PROGRAM main
VAR
    CountPulse AT %QX0.0 : BOOL;
    ResetCounter AT %QX0.1 : BOOL;
    Done AT %QX0.2 : BOOL;
    CurrentCount AT %MD0 : DINT;

    CounterInstance : CTU_DINT;
    Preset : DINT := 3;
END_VAR

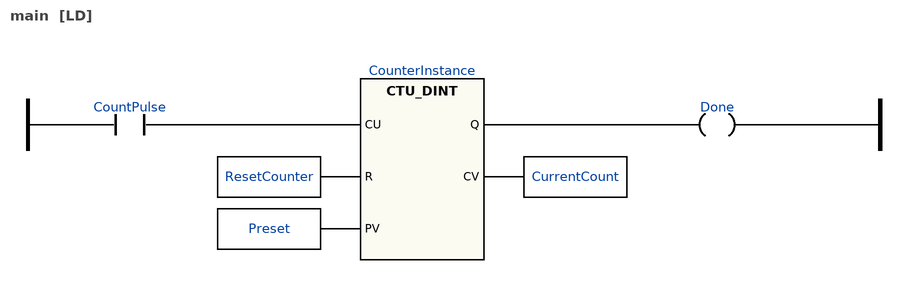
(* LD diagram, written out as Structured Text *)
CounterInstance(CU := CountPulse, R := ResetCounter, PV := Preset);
Done := CounterInstance.Q;
CurrentCount := CounterInstance.CV;
END_PROGRAM
